INTERFACE I_VirtualInputSource

PROPERTY tTimestamp : ULINT
GET
END_GET
END_PROPERTY

PROPERTY bNewData : BOOL
GET
END_GET
END_PROPERTY

END_INTERFACE

(* stored: Version 1.1.0.1
   Itf I_VirtualInputSource: Id 6e63c908-61ef-47cf-a19e-279c3212dbbb
   Property tTimestamp: Id a61af498-c2c7-43ed-9f22-15d4609e7e64
   Get Get: Id 9a55fcb5-e396-4f32-8948-a5a1af4e466e
   Property bNewData: Id 3726c995-c862-4687-8c09-8932ab7745f2
   Get Get: Id 2b9bcfab-65c3-4226-ae01-cc01198a5797 *)
